TEXTLIST LimitSwitchesTextList
  0 = 'Positive'
  1 = 'Negative'
   = ''
END_TEXTLIST

(* stored: Version 1.1.0.1, ProductVersion 3.1.4019.2
   TextList LimitSwitchesTextList: Id {7f5c8dc9-5ee0-4928-a01d-67287a79fa71} *)
